{region '#Template'}
	{attribute 'Version' := '5.0.0.0'}
	{attribute 'Tags' := '"LCID": "1031", "Text": "RA, Beleuchtung, Aktor"'}
	{attribute 'Tags' := '"LCID": "1033", "Text": "RA, Lighting, Actuator"'}
	{attribute 'Using' := '"Type": "Template", "URI": "ST_BA_LightActuatorFeedback"'}
	{attribute 'Description' := '"LCID": "1031", "Text": "Beleuchtung DALI-Aktor mit Farbtemperatur"'}
	{attribute 'Description' := '"LCID": "1033", "Text": "Lighting DALI-actuator with colour-temperature"'}
{endregion}
FUNCTION_BLOCK FB_BA_LightDALI_TC  EXTENDS FB_BA_View

VAR_INPUT
	bEn						: BOOL;						// FB-enable 
	stLightingCmd			: ST_BA_Lighting;   		// command-structure
	bInitialize				: BOOL;  					// initialize with DALI-parameters
END_VAR
VAR_OUTPUT
	bInitializing			: BOOL;						// device is being initialized
	bErr					: BOOL;						// error
	fActualLightValue		: REAL;						// actual light value
	fActualLightTemperature	: REAL;						// actual light temperature
	eActualLightPrio		: BYTE;						// actual telegram priority
	stFeedback				: ST_BA_LightActuatorFeedback;
END_VAR
VAR_INPUT CONSTANT PERSISTENT
	eAdrType				: Tc3_DALI.E_DALIAddressType	:= Tc3_DALI.E_DALIAddressType.Short;
	nAdr					: BYTE;
	nAdrRefDev				: BYTE;						// reference device if group-mode
	ipDALICommunication		: Tc3_DALI.I_DALICommunication;
END_VAR
VAR_INPUT CONSTANT
	LightActr				: FB_BA_LightActrDALI_TC;				 
	ActualLightValue		: FB_BA_AV_Op;		
END_VAR
VAR // added by the converter: edge detectors and wires of the graphical bodies
    _s1 : ST_BA_LightActuatorFeedback;
END_VAR

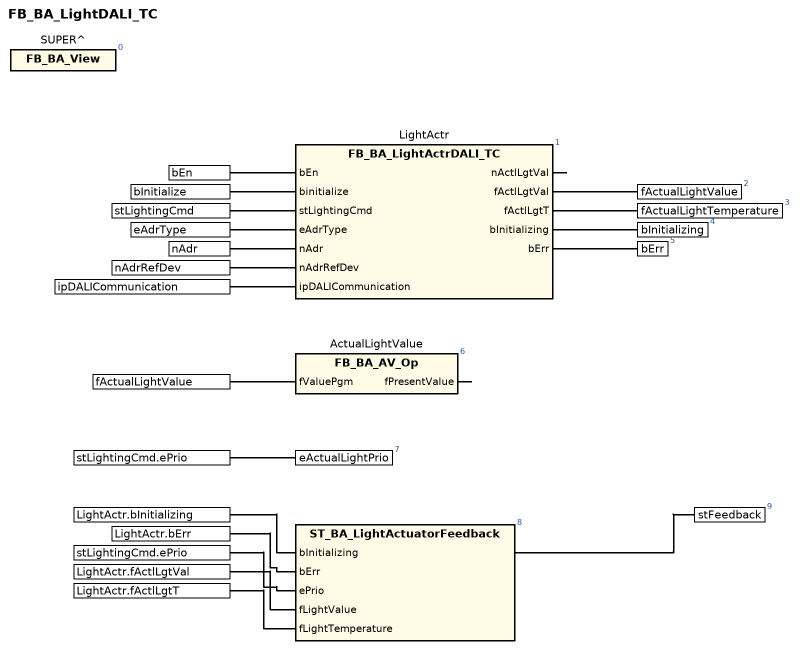
SUPER^(); // FB_BA_View
LightActr(
    bEn := bEn,
    binitialize := bInitialize,
    stLightingCmd := stLightingCmd,
    eAdrType := eAdrType,
    nAdr := nAdr,
    nAdrRefDev := nAdrRefDev,
    ipDALICommunication := ipDALICommunication); // FB_BA_LightActrDALI_TC
fActualLightValue := LightActr.fActlLgtVal;
fActualLightTemperature := LightActr.fActlLgtT;
bInitializing := LightActr.bInitializing;
bErr := LightActr.bErr;
ActualLightValue(fValuePgm := fActualLightValue); // FB_BA_AV_Op
eActualLightPrio := stLightingCmd.ePrio;
// compose _s1 : ST_BA_LightActuatorFeedback
_s1.bInitializing := LightActr.bInitializing;
_s1.bErr := LightActr.bErr;
_s1.ePrio := stLightingCmd.ePrio;
_s1.fLightValue := LightActr.fActlLgtVal;
_s1.fLightTemperature := LightActr.fActlLgtT;
stFeedback := _s1;

METHOD FB_init : BOOL
VAR_INPUT
	bInitRetains : BOOL; // if TRUE; the retain variables are initialized (warm start / cold start)
	bInCopyCode : BOOL;  // if TRUE; the instance afterwards gets moved into the copy code (online change)
END_VAR
{region 'Application parameters'}
LightActr.nHysLgtVal					:= 2;				// hysteresis to accept a new light-value-command
LightActr.fHysLgtT						:= 2;				// hysteresis to accept a new light-temperature-command
LightActr.nPrdQueryLgtVal				:= 30;				// background query light-level query
LightActr.nPrdQueryLgtT					:= 120;				// background query light-level temperature
{endregion}	
	 
{region 'Device parameters to be initially set into the device'}	
LightActr.nMinLevel						:= 126;				// DALI 1..254
LightActr.nMaxLevel						:= 254;				// DALI 1..254
LightActr.nPowerOnLevel					:= 254;				// DALI 1..254
LightActr.nSystemFailureLevel			:= 254;				// DALI 1..254
LightActr.eFadeTime						:= E_DALIFadeTime.Disabled;		
LightActr.eFadeRate						:= E_DALIFadeRate.N358StepsPerSec;		
LightActr.fTemperatureLimitWarmest		:= 2700;			// WARMEST value 0K to 1000001K
LightActr.fTemperatureLimitCoolest		:= 6500;			// COOLEST value 0K to 1000001K
LightActr.fPowerOnTemperature			:= 3000;			// 0K to 1000001K
LightActr.fSystemFailureTemperature		:= 3000;			// 0K to 1000001K
{endregion}	

{region 'BACnet'}
ActualLightValue.iParent				:= THIS^;
ActualLightValue.iLabel					:= LblFun_FeedbackLightValue;
ActualLightValue.eUnit					:= E_BA_Unit.eOther_Percent;
ActualLightValue.fCOVIncrement			:= BA2_Param.fDefCOVIncrement;	 
{endregion}
END_METHOD

END_FUNCTION_BLOCK

(* stored: Version 1.1.0.1, ProductVersion 3.1.4024.12
   POU FB_BA_LightDALI_TC: Id {bb37dc43-5701-4a8a-9955-66cb07a2333a}, SpecialFunc None
   Method FB_init: Id {fb20ad6f-d41e-4306-8582-3c79c9db63bf} *)
